// TIA Portal V20 export
// export: Created 2026-07-10T11:12:26.6400685Z, ExportSetting WithDefaults, DisplayName Totally Integrated Automation Portal, DisplayVersion V20, DisplayName TIA Portal Openness, DisplayVersion V20, DisplayName TIA Portal Version Control Interface, DisplayVersion V20, DisplayName STEP 7 Professional, DisplayVersion V20, DisplayName STEP 7 Safety, DisplayVersion V20, DisplayName WinCC Basic/Comfort/Advanced, DisplayVersion V20, DisplayName WinCC Unified, DisplayVersion V20
DATA_BLOCK "MB"   // DB1
{ S7_Optimized_Access := 'FALSE' }
VERSION : 0.1
// stored: AutoNumber false, DBAccessibleFromOPCUA true, IsOnlyStoredInLoadMemory false, IsWriteProtectedInAS false
   VAR RETAIN
      Table : Struct
         Service : Bool := FALSE;
         CycleDay : Int := 0;
         CycleStatus : Word := 16#0001;
         RestTimeC1 : UInt := 10;
         RestTimeC2 : UInt := 20;
         RestTimeC3 : UInt := 27;
         RestTimeC4 : UInt := 45;
         RestTimeC5 : UInt := 9999;
         CycleStartDay : Array[0..4] of UInt;
         LevelRCV1Min : Real := 190.0;
         LevelRCV1Max : Real := 210.0;
         LevelRCV2Min : Real := 190.0;
         LevelRCV2Max : Real := 210.0;
         LevelRCV1BasicMin : Real := 200.0;
         LevelRCV1BasicMax : Real := 250.0;
         LevelRCV2BasicMin : Real := 200.0;
         LevelRCV2BasicMax : Real := 250.0;
         LevelRCVCycle : Array[0..4] of Struct
            Min : Real;
            Max : Real;
         END_STRUCT;
         WaterCounterInPulseValue : Real := 0.1;
         WaterCounterInDailyValue : Real := 0.0;
         WaterCounterInTotalValue : Real := 0.0;
         AIOffsetCH0 : Real := 0.0;
         AIValueMinCH0 : Real := 0.0;
         AIValueMaxCH0 : Real := 1.0;
         AITimeBaseCH0 : Time := T#0MS;
         AIOffsetCH1 : Real := 0.0;
         AIValueMinCH1 : Real := 0.0;
         AIValueMaxCH1 : Real := 1200.0;
         AITimeBaseCH1 : Time := T#5MS;
         AIOffsetCH2 : Real := 0.0;
         AIValueMinCH2 : Real := 0.0;
         AIValueMaxCH2 : Real := 1200.0;
         AITimeBaseCH2 : Time := T#5MS;
         AIOffsetCH3 : Real := 0.0;
         AIValueMinCH3 : Real := 0.0;
         AIValueMaxCH3 : Real := 16.0;
         AITimeBaseCH3 : Time := T#2MS;
         AIOffsetCH4 : Real := 0.0;
         AIValueMinCH4 : Real := 0.0;
         AIValueMaxCH4 : Real := 16.0;
         AITimeBaseCH4 : Time := T#2MS;
         AIOffsetCH5 : Real := 0.0;
         AIValueMinCH5 : Real := 0.0;
         AIValueMaxCH5 : Real := 0.0;
         AITimeBaseCH5 : Time := T#0MS;
         ChlorValue : Real := 0.8276128;
         RCV1LevelValue : Real := 0.07552084;
         RCV2LevelValue : Real := 199.1832;
         WaterInPressureValue : Real := 0.0;
         WaterOutPressureValue : Real := 4.414607;
         Reserved : Real := 0.0;
         LevelRCV1AlarmMin : Real := 100.0;
         LevelRCV1AlarmMax : Real := 400.0;
         LevelRCV2AlarmMin : Real := 100.0;
         LevelRCV2AlarmMax : Real := 400.0;
         Chlor_Setpoint : Real := 0.0;
         Chlor_PulseWeight : Real := 0.0;
         Chlor_ConcentAlarm : Real := 0.9;
         Chlor_BaseDose : Real := 25.0;   // Була задача в ручному
         Chlor_SetpointMin : Real := 1.0;
         Chlor_SetpointMax : Real := 1.1;
         Chlor_Corection : Real := 0.5;
         Doser1_PulseValue : Real := 10.0;
         Reserved_2 : Int := 0;
         Reserved_3 : Int := 0;
         Doser1_DailyValue : Real := 0.0;
         Doser1_TotalValue : Real := 0.0;
         Doser1_Cunsumption : Real := 0.0;
         Doser2_PulseValue : Real := 0.81;
         Reserved_4 : Int := 0;
         Reserved_5 : Int := 0;
         Doser2_DailyValue : Real := 0.0;
         Doser2_TotalValue : Real := 0.0;
         Doser2_Cunsumption : Real := 0.0;
         PumpDoserValue : Real := 0.0;
         CalibratedPumpDoserValueMA : Real := 4.0;
         PumpDoserCalibrationMA : Real := 0.0;
         PumpDoserProductivity : Real := 6300.0;
         DampersSyncMode : Word := 16#0000;
         UsePID : Bool := FALSE;
         Damper1_PID_SetpointDeadZone : Real := 5.0;
         Damper1_PID_KP : Real := 2.0;
         Damper1_PID_KI : Real := 0.3;
         Damper1_PID_KD : Real := 0.1;
         Damper1_PID_TI : Real := 600.0;
         Damper1_PositionDeadZone : Real := 1.0;
         Damper1_FullMovingTime : Real := 26.14;
         Damper1_Position : Real := 0.0;
         Damper1_PositionSetpoint : Real := 100.0;
         Damper1_PID_Setpoint : Real := 200.0;
         Damper2_PID_SetpointDeadZone : Real := 5.0;
         Damper2_PID_KP : Real := 2.0;
         Damper2_PID_KI : Real := 0.3;
         Damper2_PID_KD : Real := 0.1;
         Damper2_PID_TI : Real := 600.0;
         Damper2_PositionDeadZone : Real := 1.0;
         Damper2_FullMovingTime : Real := 28.0;
         Damper2_Position : Real := 0.0;
         Damper2_PositionSetpoint : Real := 0.0;
         Damper2_PID_Setpoint : Real := 200.0;
         HMI_CycleOn : Bool := TRUE;
         HMI_ChlorModeOn : Bool := FALSE;
         HMI_Chlor_ChooseTank : Bool := TRUE;   // 0 - РЧВ1 1 -РЧВ2
         HMI_ManualModeOn : Bool := FALSE;
         HMI_SoundOff : Bool := TRUE;
         HMI_ManualOpenDamper1 : Bool := FALSE;
         HMI_ManualOpenDamper2 : Bool := FALSE;
         HMI_ResetWaterCounter : Bool := FALSE;
         HMI_ResetPositionDamper1 : Bool := FALSE;
         HMI_ResetPositionDamper2 : Bool := FALSE;
         HMI_StartAdjustDamper1 : Bool := FALSE;
         HMI_StartAdjustDamper2 : Bool := FALSE;
         HMI_StopAdjustDamper1 : Bool := FALSE;
         HMI_StopAdjustDamper2 : Bool := FALSE;
         HMI_WeightToZero : Bool := FALSE;
         HMI_WeightAlarmReset : Bool := FALSE;
         Alarms_Open1 : Bool := FALSE;
         Alarms_Open2 : Bool := FALSE;
         Alarms_ChlorLargeConsumption : Bool := FALSE;
         Alarms_RCV1Max : Bool := FALSE;
         Alarms_RCV1Min : Bool := TRUE;
         Alarms_RCV2Max : Bool := FALSE;
         Alarms_RCV2Min : Bool := FALSE;
         Alarms_RCV1Error : Bool := FALSE;
         Alarms_RCV2Error : Bool := FALSE;
         Alarms_ChlorMax : Bool := FALSE;
         Alarms_NoFlow : Bool := FALSE;
         Alarms_WaterOutMax : Bool := FALSE;
         Alarms_WaterOutMin : Bool := FALSE;
         Alarms_NoPowerSupply : Bool := FALSE;
         Alarms_WaterInMax : Bool := FALSE;
         Alarms_WaterInMin : Bool := FALSE;
         WaterOutMaxValue : Real := 6.0;
         WaterOutMinValue : Real := 1.5;
         WaterOutAlarmTime : DInt := 10;
         GlobalAlarm : Bool := FALSE;
         SensorWeightVoltage1 : Real := 1.681112;
         WeightValueMin1 : Real := 356.0;
         WeightValueMax1 : Real := 361.0;
         WeightValueOffset1 : Real := 0.0;
         WeightValue1 : Real := 353.3342;
         WeightVoltageMin1 : Real := 1.691255;
         WeightVoltageMax1 : Real := 1.71028;
         DayChangeFlag : Bool := TRUE;
         Damper1_AdjustBusy : Bool := FALSE;
         Damper1_AdjustError : Bool := FALSE;
         Damper1_AdjustDone : Bool := FALSE;
         Damper2_AdjustBusy : Bool := FALSE;
         Damper2_AdjustError : Bool := FALSE;
         Damper2_AdjustDone : Bool := FALSE;
         "Damper1_Close/Open" : Bool := FALSE;
         "Damper2_Close/Open" : Bool := FALSE;
         "Damper1_Manual/Auto" : Bool := FALSE;
         "Damper2_Manual/Auto" : Bool := TRUE;
         SensorWeightVoltage2 : Real := -0.2375481;
         WeightValueMin2 : Real := 0.0;
         WeightValueMax2 : Real := 5.0;
         WeightValueOffset2 : Real := 0.0;
         WeightValue2 : Real := 0.0;
         WeightVoltageMin2 : Real := 0.155;
         WeightVoltageMax2 : Real := 0.177;
         WaterConsumption : Real := 0.0;
         LevelRCV1AlarmMinBasic : Real := 0.0;
         LevelRCV1AlarmMaxBasic : Real := 0.0;
         LevelRCV2AlarmMinBasic : Real := 0.0;
         LevelRCV2AlarmMaxBasic : Real := 0.0;
         LevelRCV1AlarmDeltaC1 : Real := 20.0;
         LevelRCV1AlarmDeltaC2 : Real := 20.0;
         LevelRCV1AlarmDeltaC3 : Real := 20.0;
         LevelRCV1AlarmDeltaC4 : Real := 20.0;
         LevelRCV1AlarmDeltaC5 : Real := 20.0;
         LevelRCV2AlarmDeltaC1 : Real := 20.0;
         LevelRCV2AlarmDeltaC2 : Real := 20.0;
         LevelRCV2AlarmDeltaC3 : Real := 20.0;
         LevelRCV2AlarmDeltaC4 : Real := 20.0;
         LevelRCV2AlarmDeltaC5 : Real := 20.0;
         WaterInPresMaxValue : Real := 8.0;
         WaterInPresMinValue : Real := 1.5;
         WaterInPresAlarmTime : DInt := 10;
         EndTag : Real := 0.0;
         WeightingEnable : Bool := TRUE;
         WeightingSetZero : Bool := FALSE;
         WeightValue1Liters : Real := 294.4452;
         WeightValue2Liters : Real := 0.0;
         WeightSensor1Error : Bool := FALSE;
         WeightSensor2Error : Bool := FALSE;
         Weighting_SaveManualValue : Bool := FALSE;
         Weighting_ManualValue1 : Real := 0.0;
         Weighting_ManualValue2 : Real := 0.0;
         WeightingDelay : DInt := 0;
         WeightingDeadZone : Real := 0.0;
         WeightingStat_CalendarMonth : Array[1..30] of UInt;
         WeightingStat_CalendarDay : Array[1..30] of UInt;
         WeightingStat_DayCycle : Array[1..30] of Int;
         WeightingStat_Counsumed1 : Array[1..30] of Real;
         WeightingStat_Load1 : Array[1..30] of Real;
         WeightingStat_Counsumed2 : Array[1..30] of Real;
         WeightingStat_Load2 : Array[1..30] of Real;
         ChlorReg_Update : Bool := FALSE;
         ChlorReg_DateTime : DTL := DTL#1970-01-01-00:00:00;
         HMI_ChlorReg_ValueRCV : Real := 0.0;
         HMI_ChlorReg_ValuePt : Real := 0.0;
         ChlorReg_ChlorValueRCV : Real := 0.0;
         ChlorReg_ChlorValuePt : Real := 0.0;
         ChlorReg_Age : Int := 0;
         Reserved_1 : Int := 0;
         ChlorReg_AgeF : Real := 0.0;
         WaterCounterIn_DailyCount : DInt := 0;
         WaterCounterIn_TotalCount : DInt := 0;
         Doser1_DailyPulses : DInt := 0;
         Doser1_TotalPulses : DInt := 0;
         Doser2_DailyPulses : DInt := 0;
         Doser2_TotalPulses : DInt := 0;
         WaterTemperature : Real := 18.22104;
         ChlorConsumptionTable : Array[0..3] of Struct
            Day : Int;
            MonitorTIme : Real;
            Consumption : Real;
         END_STRUCT;
         DoserNotWork : Bool := FALSE;
         Chlor_AutoMode : Bool := TRUE;
         Chlor_StartManual : Bool := FALSE;
         Chloration_ChooseCounter : Bool := FALSE;
         RecerculationFlow : Real := 0.0;
         FlowWithouRecerculation : Real := 17.51287;
         ChlorationParams : Struct
            SetpointMin : Real := 0.0;
            SetpointMax : Real := 0.0;
            BaseDose : Real := 0.0;
            ActualDose : Real := 0.0;
            DoseChangeMax : Real := 25.0;
            DosingMin : Real := 0.0;
            DosingMax : Real := 35.0;
            CorectionCoef : Real := 1.0;
         END_STRUCT;
         ChangeChlorMeasure : Bool := FALSE;
         MeasureChanged : Bool := FALSE;
         CriticalMeasureON : Bool := FALSE;
         MeasureNotEntered : Bool := FALSE;
         ChlorationCounter_SwitchOn : Bool := FALSE;
         ChlorMeasuredValue : Real := 0.0;
         ChlorMeasureTable : Array[0..3] of Struct
            CycleDay : Int;
            MeasureTime : Real;
            BlockTime : Real;
         END_STRUCT;
         TimeToMeasure : Real := 1.0;
         TimeToBlock : Real := 29.0;
         CriticalMeasure : Real := 1.5;
         Chlor_PulseWeight_1 : Real := 1.0;
         Chlor_ManualSetpoint_1 : Real := 0.0;
         MeasuredChlor : Real := 0.0;
         ClO2 : Struct
            AbsoluteDosing : Real := 0.0;
            ProportionalDosingEmbedded : Real := 0.0;
            ProportionalDosingExternal : Real := 0.0;
            ChooseDosing : Word := 16#1204;
            DosersActive : Word := 16#0006;
            WorkMode : Word := 16#0001;
            Doser1Productivity : Real := 0.0;
            Doser2Productivity : Real := 0.0;
            Pressure : Real := 0.0;
            SystemProductivity : Real := 0.0;
            Alarms : Word := 16#0000;
         END_STRUCT;
         WaterCounterOut_DailyCount : DInt := 3;
         WaterCounterOut_TotalCount : DInt := 3;
         WaterCounterOut_DailyValue : Real := 0.3;
         WaterCounterOut_TotalValue : Real := 0.3;
         WaterCounterOut_PulseValue : Real := 0.1;
         WaterCounterOut_Consumption : Real := 16#7F80_0000;
         ChlorationCounter_SwitchDay : Int := 5;
         END : Array[0..10] of Word;
      END_STRUCT;
   END_VAR
BEGIN
   Table.CycleStartDay[0] := 0;
   Table.CycleStartDay[1] := 10;
   Table.CycleStartDay[2] := 20;
   Table.CycleStartDay[3] := 27;
   Table.CycleStartDay[4] := 45;
   Table.LevelRCVCycle[0].Min := 190.0;
   Table.LevelRCVCycle[1..3].Min := 270.0;
   Table.LevelRCVCycle[4].Min := 190.0;
   Table.LevelRCVCycle[0].Max := 210.0;
   Table.LevelRCVCycle[1..3].Max := 310.0;
   Table.LevelRCVCycle[4].Max := 210.0;
   Table.WeightingStat_CalendarMonth[1] := 7;
   Table.WeightingStat_CalendarMonth[2..30] := 0;
   Table.WeightingStat_CalendarDay[1] := 7;
   Table.WeightingStat_CalendarDay[2..30] := 0;
   Table.WeightingStat_DayCycle[1..30] := 0;
   Table.WeightingStat_Counsumed1[1] := 0.0133667;
   Table.WeightingStat_Counsumed1[2..30] := 0.0;
   Table.WeightingStat_Load1[1] := 353.3476;
   Table.WeightingStat_Load1[2..30] := 0.0;
   Table.WeightingStat_Counsumed2[1..30] := 0.0;
   Table.WeightingStat_Load2[1..30] := 0.0;
   Table.ChlorConsumptionTable[0].Day := 0;
   Table.ChlorConsumptionTable[1].Day := 6;
   Table.ChlorConsumptionTable[2].Day := 18;
   Table.ChlorConsumptionTable[3].Day := 30;
   Table.ChlorConsumptionTable[0..3].MonitorTIme := 1.0;
   Table.ChlorConsumptionTable[0..3].Consumption := 3.0;
   Table.ChlorMeasureTable[0..3].CycleDay := 0;
   Table.ChlorMeasureTable[0..3].MeasureTime := 1.0;
   Table.ChlorMeasureTable[0..3].BlockTime := 29.0;
   Table.END[0..10] := 16#0000;
END_DATA_BLOCK
